INTERFACE I_Deserializable EXTENDS __SYSTEM.IQueryInterface

METHOD TryDeserializeFrom : BOOL
VAR_INPUT
	Deserializer : I_Deserializer;
	Feedback : I_DeserializerFeedback;
END_VAR
END_METHOD

END_INTERFACE

(* stored: Version 1.1.0.1, ProductVersion 3.1.4024.12
   Itf I_Deserializable: Id {ecdccc31-31bd-0587-113d-42d1fa3ffec3}
   Method TryDeserializeFrom: Id {ef7fd094-25e7-073b-3cc2-f6394ba9b470} *)
